TYPE (* IEC 61131-3-2.3.3.2 *)
  (* Standard: 61131-3 *)
  (* Version 0.3, 2001-03-02, JHC, Rockwell Automation, Test revised Java code generation. *)
  (* Version 0.2, 2000-05-16, JHC, Rockwell Automation, File type changed to ".dtp" *)
  (* Version 0.1, 2000-05-10, JHC, Rockwell Automation, Corrected encoding of values. *)
  (* Compiler header: package fb.rt.ita; *)
  (* Compiler Java IBM VisualAge 3.0 *)
  (* ASN.1 tag PRIVATE 11 *)
  ANALOG_SIGNAL_RANGE : (
    BIPOLAR_10V, (* -10 to+10 VDC *)
    UNIPOLAR_10V, (* 0 to+10 VDC *)
    UNIPOLAR_1_5V, (* +1 to+5 VDC *)
    UNIPOLAR_0_5V, (* 0 to+5 VDC *)
    UNIPOLAR_4_20_MA, (* +4 to+20 mADC *)
    UNIPOLAR_0_20_MA (* 0 to+20 mADC *)
  ) := UNIPOLAR_1_5V;
END_TYPE
